Yaskawa INFORM job: UF-STATION-2-REF.JBI

/JOB
//NAME UF-STATION-2-REF
//POS
///NPOS 3,0,0,1,0,0
///TOOL 1
///POSTYPE PULSE
///PULSE
C00000=236239,16978,-17785,155524,-149241,-118719
C00001=314364,28931,49876,93809,-165788,-92057
C00002=314361,28777,49430,93786,-165625,-92181
P01600=314361,28777,49430,93786,-165625,-92181
//INST
///DATE 2018/09/17 11:56
///ATTR SC,RW
///GROUP1 RB1
///LVARS 0,0,0,0,0,10,0,0
NOP
REFP 1 C00000
REFP 2 C00001
REFP 3 C00002
GETS PX1600 $PX011
SET LP000 P1600
GETS PX1600 $PX012
SET LP001 P1600
GETS PX1600 $PX013
SET LP002 P1600
MFRAME UF#(12) LPX000 LPX001 LPX002
END
